# EPICS substitutions: RadiationMonitoringApp/Db/common/mams-station.substitutions
file ams-printer.template
{
     pattern { P,                PORT     }
             { AMS:SITE:$(UNIT), $(APORT) }
}
